Staubli VAL3: start.pgx

program start()
begin
  //nMoveType:
  //0:Frame
  //1:tool
  //2:joint
  taskCreateSync "vel",0.004,bSync,setVel(nMoveType,world,tTool,mNominal,nVelCmd)
end
